// Reads a string field value from the input.
FUNCTION F_ReadString : HRESULT
VAR_INPUT CONSTANT
    aBuffer : ARRAY [*] OF BYTE;   
END_VAR
VAR_IN_OUT
    stState : ST_ParserInternalState;
END_VAR
VAR_INPUT
    anyStringOut : ANY_STRING;
END_VAR
VAR
    nStrLength : UDINT;
END_VAR

F_ReadString := S_OK;

F_ReadString := F_ParseLength(aBuffer, stState, nLength=> nStrLength);
IF FAILED(F_ReadString) THEN
    RETURN;
END_IF

F_ReadString := F_ReadRawString(aBuffer, nStrLength, F_ToAnyType(anyStringOut), stState);

END_FUNCTION

(* stored: Version 1.1.0.1
   POU F_ReadString: Id {d90e99f7-a7ef-43ab-94c0-307afbb7fd5d}, SpecialFunc None *)
